TYPE ST_PackageInfo :
STRUCT
	PackageLength: UDINT;
	MessageType: USINT;
END_STRUCT
END_TYPE

(* stored: Version 1.1.0.1, ProductVersion 3.1.4020.12
   DUT ST_PackageInfo: Id {3b435365-bc0b-4660-820d-56ee31694968} *)
